FUNCTION_BLOCK SelectMode (* Basic Function Block Type *)
  (* Standard: 61499-2 *)
  (* Version 0.0, 2/18/2024, midxav, Template *)
  PACKAGE Main;
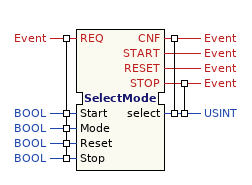
  EVENT_INPUT
    REQ WITH Start, Mode, Reset, Stop; (* Normal Execution Request *)
  END_EVENT
  EVENT_OUTPUT
    CNF WITH select; (* Execution Confirmation *)
    START;
    RESET;
    STOP WITH select;
  END_EVENT
  VAR_INPUT
    Start : BOOL;
    Mode : BOOL; (* Input event qualifier *)
    Reset : BOOL;
    Stop : BOOL;
  END_VAR
  VAR_OUTPUT
    select : USINT; (* Output event qualifier *)
  END_VAR
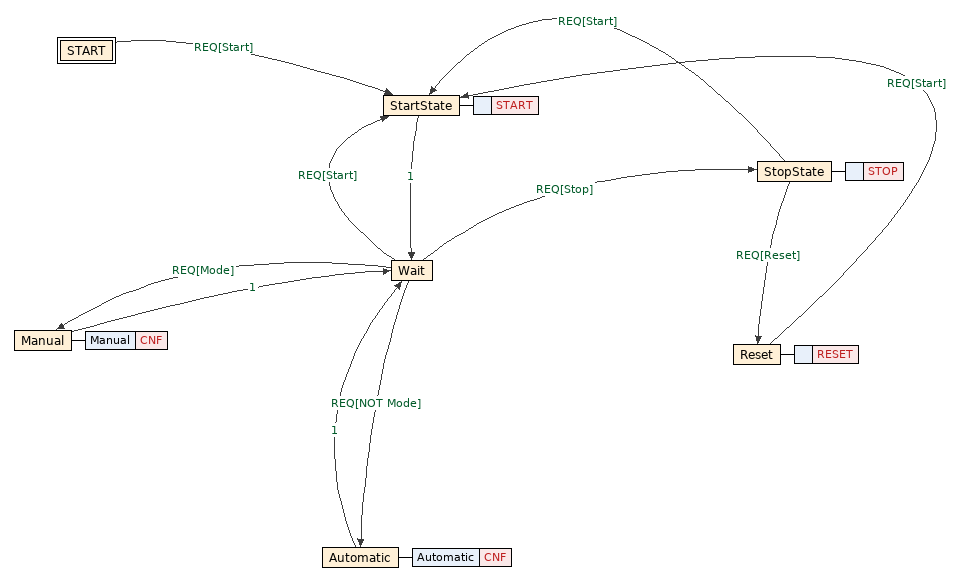
  EC_STATES
    START; (* Initial State *)
    Manual : Manual -> CNF; (* Normal execution *)
    Automatic : Automatic -> CNF;
    Reset : -> RESET;
    StopState : -> STOP;
    Wait;
    StartState : -> START;
  END_STATES
  EC_TRANSITIONS
    Wait TO Manual := REQ[Mode];
    Manual TO Wait := 1;
    Wait TO Automatic := REQ[NOT Mode];
    Automatic TO Wait := 1;
    START TO StartState := REQ[Start];
    Wait TO StopState := REQ[Stop];
    StopState TO Reset := REQ[Reset];
    StopState TO StartState := REQ[Start];
    Reset TO StartState := REQ[Start];
    StartState TO Wait := 1;
    Wait TO StartState := REQ[Start];
  END_TRANSITIONS
  ALGORITHM INIT IN ST: (* Initialization algorithm *)
;
  END_ALGORITHM
  ALGORITHM Manual IN ST: (* Normally executed algorithm *)
select := 0;
  END_ALGORITHM
  ALGORITHM Automatic IN ST:
select := 1;
  END_ALGORITHM
END_FUNCTION_BLOCK
